// SIMATIC STEP 7 (V5.x) project ZEn01_08_STEP7__Mix
// CPU: CPU314(1)
// station: Hardware
// station: SIMATIC 300(1)
// program: S7-Program(1)

SYMBOL_TABLE
"DB_feed_pump_A"	DB 1	FB 1	// Instance DB for controlling feed pump A
"DB_feed_pump_B"	DB 2	FB 1	// Instance DB for controlling feed pump B
"DB_agitator"	DB 3	FB 1	// Instance DB for controlling agitator motor
"Motor_block"	FB 1	FB 1	// FB for controlling pumps and agitator motor
"Valve_block"	FC 1	FC 1	// FC for controlling valves
"Feed_pump_A_start"	I 0.0	BOOL	// Start pushbutton feed pump for ingredient A
"Feed_pump_A_stop"	I 0.1	BOOL	// Stop pushbutton feed pump for ingredient A
"Flow_A"	I 0.2	BOOL	// Ingredient A flows
"Feed_pump_B_start"	I 0.3	BOOL	// Start pushbutton feed pump for ingredient B
"Feed_pump_B_stop"	I 0.4	BOOL	// Stop pushbutton feed pump for ingredient B
"Flow_B"	I 0.5	BOOL	// Ingredient B flows
"Drain_open"	I 0.6	BOOL	// Pushbutton for opening drain valve
"Drain_closed"	I 0.7	BOOL	// Pushbutton for closing drain valve
"Agitator_running"	I 1.0	BOOL	// Feedback signal from the agitator motor
"Agitator_start"	I 1.1	BOOL	// Start pushbutton agitator
"Agitator_stop"	I 1.2	BOOL	// Stop pushbutton agitator
"Tank_below_max"	I 1.3	BOOL	// Sensor "Mixing tank not full"
"Tank_above_min"	I 1.4	BOOL	// Sensor "Mixing tank above minimum level"
"Tank_not_empty"	I 1.5	BOOL	// Sensor "Mixing tank not empty"
"EMER_STOP_off"	I 1.6	BOOL	// EMERGENCY STOP switch
"Reset_maint"	I 1.7	BOOL	// Reset pushbutton for maintenance display (all motors)
"Inlet_valve_A"	Q 4.0	BOOL	// Activates the inlet valve for ingredient A
"Feed_valve_A"	Q 4.1	BOOL	// Activates the feed valve for ingredient A
"Feed_pump_A_on"	Q 4.2	BOOL	// Display lamp for "Feed pump ON ingredient A"
"Feed_pump_A_off"	Q 4.3	BOOL	// Display lamp for "Feed pump OFF ingredient A"
"Feed_pump_A"	Q 4.4	BOOL	// Activates the feed pump for ingredient A
"Feed_pump_A_fault"	Q 4.5	BOOL	// Display lamp for "Feed pump A fault"
"Feed_pump_A_maint"	Q 4.6	BOOL	// Display lamp for "Feed pump A maintenance"
"Inlet_valve_B"	Q 5.0	BOOL	// Activates the inlet valve for ingredient B
"Feed_valve_B"	Q 5.1	BOOL	// Activates the feed valve for ingredient B
"Feed_pump_B_on"	Q 5.2	BOOL	// Display lamp for "Feed pump ON ingredient B"
"Feed_pump_B_off"	Q 5.3	BOOL	// Display lamp for "Feed pump OFF ingredient B"
"Feed_pump_B"	Q 5.4	BOOL	// Activates the feed pump for ingredient B
"Feed_pump_B_fault"	Q 5.5	BOOL	// Display lamp for "Feed pump B fault"
"Feed_pump_B_maint"	Q 5.6	BOOL	// Display lamp for "Feed pump B maintenance"
"Agitator"	Q 8.0	BOOL	// Activates the agitator
"Agitator_on"	Q 8.1	BOOL	// Display lamp for "Agitator ON"
"Agitator_off"	Q 8.2	BOOL	// Display lamp for "Agitator OFF"
"Agitator_fault"	Q 8.3	BOOL	// Display lamp for "Agitator motor fault"
"Agitator_maint"	Q 8.4	BOOL	// Display lamp for "Agitator motor maintenance"
"Tank_max_disp"	Q 9.0	BOOL	// Display lamp for "Mixing tank full"
"Tank_min_disp"	Q 9.1	BOOL	// Display lamp for "Mixing tank below minimum level"
"Tank_empty_disp"	Q 9.2	BOOL	// Display lamp for "Mixing tank empty"
"Drain"	Q 9.5	BOOL	// Activates the drain valve
"Drain_open_disp"	Q 9.6	BOOL	// Display lamp for "Drain valve open"
"Drain_closed_disp"	Q 9.7	BOOL	// Display lamp for "Drain valve closed"
END_SYMBOL_TABLE

FUNCTION_BLOCK "Motor_block"	// FB 1
VERSION : 0.0
VAR_INPUT
  Start : BOOL ;
  Stop : BOOL ;
  Response : BOOL ;
  Reset_Maint : BOOL ;
  Timer_No : TIMER ;
  Response_Time : S5TIME ;
END_VAR
VAR_OUTPUT
  Fault : BOOL ;
  Start_Dsp : BOOL ;
  Stop_Dsp : BOOL ;
  Maint : BOOL ;
END_VAR
VAR_IN_OUT
  Motor : BOOL ;
END_VAR
VAR
  Time_bin : WORD ;
  Time_BCD : WORD ;
  Starts : INT ;
  Start_Edge : BOOL ;
END_VAR
BEGIN
NETWORK
TITLE = Start/Stop and Latching
      A(;
      O     #Start;
      O     #Motor;
      );
      AN    #Stop;
      =     #Motor;
NETWORK
TITLE = Startup Monitoring
// (network holds code this reader does not know; not shown)
NETWORK
TITLE = Start Lamp / Fault Reset
      A     #Response;
      =     #Start_Dsp;
      R     #Fault;
NETWORK
TITLE = Stop Lamp
      AN    #Response;
      =     #Stop_Dsp;
NETWORK
TITLE = Count Starts
      A     #Motor;
      FP    #Start_Edge;
      JCN   lab1;
      L     #Starts;
      +     1;
      T     #Starts;
lab1: NOP   0;
NETWORK
TITLE = Maintenance
      L     #Starts;
      L     50;
      >=I;
      =     #Maint;
NETWORK
TITLE = Reset Maintenance
      A     #Reset_Maint;
      A     #Maint;
      JCN   END;
      L     0;
      T     #Starts;
END:  NOP   0;
END_FUNCTION_BLOCK

FUNCTION "Valve_block" : VOID	// FC 1
VERSION : 0.0
VAR_INPUT
  Open : BOOL ;
  Close : BOOL ;
END_VAR
VAR_OUTPUT
  Dsp_Open : BOOL ;
  Dsp_Closed : BOOL ;
END_VAR
VAR_IN_OUT
  Valve : BOOL ;
END_VAR
BEGIN
NETWORK
TITLE = Open/Close and Latching
      A(;
      O     #Open;
      O     #Valve;
      );
      AN    #Close;
      =     #Valve;
NETWORK
TITLE = Display "Valve open"
      A     #Valve;
      =     #Dsp_Open;
NETWORK
TITLE = Display "Valve closed"
      AN    #Valve;
      =     #Dsp_Closed;
END_FUNCTION

DATA_BLOCK "DB_feed_pump_A"	// DB 1
VERSION : 0.0
"Motor_block"
BEGIN
END_DATA_BLOCK

DATA_BLOCK "DB_feed_pump_B"	// DB 2
VERSION : 0.0
"Motor_block"
BEGIN
END_DATA_BLOCK

DATA_BLOCK "DB_agitator"	// DB 3
VERSION : 0.0
"Motor_block"
BEGIN
END_DATA_BLOCK

ORGANIZATION_BLOCK OB 1
VERSION : 0.0
VAR_TEMP
  OB1_EV_CLASS : BYTE ;	//Bits 0-3 = 1 (Coming event), Bits 4-7 = 1 (Event class 1)
  OB1_SCAN_1 : BYTE ;	//1 (Cold restart scan 1 of OB1), 3 (Scan 2-n of OB1)
  OB1_PRIORITY : BYTE ;	//1 (Priority of 1 is lowest)
  OB1_OB_NUMBR : BYTE ;	//1 (Organization block 1, OB1)
  OB1_RESERVED_1 : BYTE ;	//Reserved for system
  OB1_RESERVED_2 : BYTE ;	//Reserved for system
  OB1_PREV_CYCLE : INT ;	//Cycle time of previous OB1 scan (milliseconds)
  OB1_MIN_CYCLE : INT ;	//Minimum cycle time of OB1 (milliseconds)
  OB1_MAX_CYCLE : INT ;	//Maximum cycle time of OB1 (milliseconds)
  OB1_DATE_TIME : DATE_AND_TIME ;	//Date and time OB1 started
  Enable_Motor : BOOL ;
  Enable_Valve : BOOL ;
  Start_Fulfilled : BOOL ;
  Stop_Fulfilled : BOOL ;
  Inlet_Valve_A_Open : BOOL ;
  Inlet_Valve_A_Closed : BOOL ;
  Feed_Valve_A_Open : BOOL ;
  Feed_Valve_A_Closed : BOOL ;
  Inlet_Valve_B_Open : BOOL ;
  Inlet_Valve_B_Closed : BOOL ;
  Feed_Valve_B_Open : BOOL ;
  Feed_Valve_B_Closed : BOOL ;
  Open_Drain : BOOL ;
  Close_Drain : BOOL ;
  Close_Valve_Fulfilled : BOOL ;
END_VAR
BEGIN
NETWORK
TITLE = Interlock for Feed Pump A
      A     "EMER_STOP_off";
      A     "Tank_below_max";
      AN    "Drain";
      =     #Enable_Motor;
NETWORK
TITLE = Call FB Motor for Ingredient A
      A     "Feed_pump_A_start";
      A     #Enable_Motor;
      =     #Start_Fulfilled;
      A(;
      O     "Feed_pump_A_stop";
      ON    #Enable_Motor;
      );
      =     #Stop_Fulfilled;
      CALL  "Motor_block" , "DB_feed_pump_A" (
           Start                    := #Start_Fulfilled,
           Stop                     := #Stop_Fulfilled,
           Response                 := "Flow_A",
           Reset_Maint              := "Reset_maint",
           Timer_No                 := T 12,
           Response_Time            := 1792,
           Fault                    := "Feed_pump_A_fault",
           Start_Dsp                := "Feed_pump_A_on",
           Stop_Dsp                 := "Feed_pump_A_off",
           Maint                    := "Feed_pump_A_maint",
           Motor                    := "Feed_pump_A");
NETWORK
TITLE = Delay Valve Enable Ingredient A
      A     "Feed_pump_A";
      L     S5T#1S;
      SD    T 13;
      AN    "Feed_pump_A";
      R     T 13;
      A     T 13;
      =     #Enable_Valve;
NETWORK
TITLE = Inlet Valve Control for Ingredient A
      AN    "Flow_A";
      AN    "Feed_pump_A";
      =     #Close_Valve_Fulfilled;
      CALL  "Valve_block" (
           Open                     := #Enable_Valve,
           Close                    := #Close_Valve_Fulfilled,
           Dsp_Open                 := #Inlet_Valve_A_Open,
           Dsp_Closed               := #Inlet_Valve_A_Closed,
           Valve                    := "Inlet_valve_A");
NETWORK
TITLE = Feed Valve Control for Ingredient A
      AN    "Flow_A";
      AN    "Feed_pump_A";
      =     #Close_Valve_Fulfilled;
      CALL  "Valve_block" (
           Open                     := #Enable_Valve,
           Close                    := #Close_Valve_Fulfilled,
           Dsp_Open                 := #Feed_Valve_A_Open,
           Dsp_Closed               := #Feed_Valve_A_Closed,
           Valve                    := "Feed_valve_A");
NETWORK
TITLE = Interlock for Feed Pump B
      A     "EMER_STOP_off";
      A     "Tank_below_max";
      AN    "Drain";
      =     #Enable_Motor;
NETWORK
TITLE = Call FB Motor for Ingredient B
      A     "Feed_pump_B_start";
      A     #Enable_Motor;
      =     #Start_Fulfilled;
      A(;
      O     "Feed_pump_B_stop";
      ON    #Enable_Motor;
      );
      =     #Stop_Fulfilled;
      CALL  "Motor_block" , "DB_feed_pump_B" (
           Start                    := #Start_Fulfilled,
           Stop                     := #Stop_Fulfilled,
           Response                 := "Flow_B",
           Reset_Maint              := "Reset_maint",
           Timer_No                 := T 14,
           Response_Time            := 1792,
           Fault                    := "Feed_pump_B_fault",
           Start_Dsp                := "Feed_pump_B_on",
           Stop_Dsp                 := "Feed_pump_B_off",
           Maint                    := "Feed_pump_B_maint",
           Motor                    := "Feed_pump_B");
NETWORK
TITLE = Delay Valve Enable Ingredient B
      A     "Feed_pump_B";
      L     S5T#1S;
      SD    T 15;
      AN    "Feed_pump_B";
      R     T 15;
      A     T 15;
      =     #Enable_Valve;
NETWORK
TITLE = Inlet Valve Control for Ingredient B
      AN    "Flow_B";
      AN    "Feed_pump_B";
      =     #Close_Valve_Fulfilled;
      CALL  "Valve_block" (
           Open                     := #Enable_Valve,
           Close                    := #Close_Valve_Fulfilled,
           Dsp_Open                 := #Inlet_Valve_B_Open,
           Dsp_Closed               := #Inlet_Valve_B_Closed,
           Valve                    := "Inlet_valve_B");
NETWORK
TITLE = Feed Valve Control for Ingredient B
      AN    "Flow_B";
      AN    "Feed_pump_B";
      =     #Close_Valve_Fulfilled;
      CALL  "Valve_block" (
           Open                     := #Enable_Valve,
           Close                    := #Close_Valve_Fulfilled,
           Dsp_Open                 := #Feed_Valve_B_Open,
           Dsp_Closed               := #Feed_Valve_B_Closed,
           Valve                    := "Feed_valve_B");
NETWORK
TITLE = Interlock for Agitator
      A     "EMER_STOP_off";
      A     "Tank_above_min";
      AN    "Drain";
      =     #Enable_Motor;
NETWORK
TITLE = Call FB Motor for Agitator
      A     "Agitator_start";
      A     #Enable_Motor;
      =     #Start_Fulfilled;
      A(;
      O     "Agitator_stop";
      ON    #Enable_Motor;
      );
      =     #Stop_Fulfilled;
      CALL  "Motor_block" , "DB_agitator" (
           Start                    := #Start_Fulfilled,
           Stop                     := #Stop_Fulfilled,
           Response                 := "Agitator_running",
           Reset_Maint              := "Reset_maint",
           Timer_No                 := T 16,
           Response_Time            := 4352,
           Fault                    := "Agitator_fault",
           Start_Dsp                := "Agitator_on",
           Stop_Dsp                 := "Agitator_off",
           Maint                    := "Agitator_maint",
           Motor                    := "Agitator");
NETWORK
TITLE = Interlock for Drain Valve
      A     "EMER_STOP_off";
      A     "Tank_not_empty";
      AN    "Agitator";
      =     #Enable_Valve;
NETWORK
TITLE = Drain Valve Control
      A     "Drain_open";
      A     #Enable_Valve;
      =     #Open_Drain;
      A(;
      O     "Drain_closed";
      ON    #Enable_Valve;
      );
      =     #Close_Drain;
      CALL  "Valve_block" (
           Open                     := #Open_Drain,
           Close                    := #Close_Drain,
           Dsp_Open                 := "Drain_open_disp",
           Dsp_Closed               := "Drain_closed_disp",
           Valve                    := "Drain");
NETWORK
TITLE = Container Level Display
      AN    "Tank_below_max";
      =     "Tank_max_disp";
      AN    "Tank_above_min";
      =     "Tank_min_disp";
      AN    "Tank_not_empty";
      =     "Tank_empty_disp";
END_ORGANIZATION_BLOCK
